INTERFACE I_Collection EXTENDS __SYSTEM.IQueryInterface

PROPERTY Count : UDINT
GET
END_GET
END_PROPERTY

END_INTERFACE

(* stored: Version 1.1.0.1, ProductVersion 3.1.4024.9
   Itf I_Collection: Id {9f6303c3-5dbf-423d-a223-eb75585587db}
   Property Count: Id {e95f9f46-aba8-4a54-9ebb-cdbb7d350f3a}
   Get Get: Id {7f219083-c12f-4dd0-a221-110fdeaca3ab} *)
